{attribute 'qualified_only'}
{attribute 'strict'}
TYPE E_SlitPairStates :
(
    eStartup := 0,
    eInit,
    eInitGearOutCheck,
    eCheckHomeStatus,
    eHomeBlades,
    eCheckBladeHomeComplete,
    eHomeGap,
    eCheckGapHomeComplete,
    eGearInSlits,
    eCheckGearInSlitsComplete,
    eSlitsOperational,
    eGearOutBlades,
    eCheckGearOutComplete,
    eResetCalibration,
    eError,
    eErrorGearOut,
    eErrorGearOutCheck,
    eErrorResetAxes,
    eErrorResetCheck
) UDINT;
END_TYPE

(* stored: Version 1.1.0.1
   DUT E_SlitPairStates: Id {bd1cffbb-4918-4a16-817e-cea08bf2daf5} *)
